INTERFACE I_AlarmActions

METHOD Acknowledge : I_AlarmActionBy
VAR_INPUT
END_VAR
END_METHOD

METHOD Deactivate : I_AlarmActionBy
VAR_INPUT
END_VAR
END_METHOD

METHOD Raise : I_AlarmActionBy
VAR_INPUT
END_VAR
END_METHOD

END_INTERFACE

(* stored: Version 1.1.0.1, ProductVersion 3.1.4024.14
   Itf I_AlarmActions: Id {78311afd-5039-09e9-2e01-ec212a338902}
   Method Acknowledge: Id {27cadfb9-70a1-0f63-1fa5-1c36d13f7186}
   Method Deactivate: Id {4b0cc508-0a65-0c13-0908-4c5fa0752ee4}
   Method Raise: Id {350c0da9-4251-06d5-39cb-5a5af1876fd3} *)
